INTERFACE ITF_CyclicUpdate

// Uses HRESULT outputs for management of different scenarios, such as errors and non-completes

//    0 - No Output / Execute In Progress
//    1 - Execute Complete
//    2 - Execute Failed, No Program Error, Object's Internal Timer Exceeded Limit.
//   -1 - Execute Failed, Program Error

METHOD CyclicUpdate : HRESULT

// Uses HRESULT outputs for management of different scenarios, such as errors and non-completes

//    0 - No Output / Execute In Progress
//    1 - Execute Complete
//    2 - Execute Failed, No Program Error, Object's Internal Timer Exceeded Limit.
//   -1 - Execute Failed, Program Error
END_METHOD

END_INTERFACE

(* stored: Version 1.1.0.1, ProductVersion 3.1.4024.12
   Itf ITF_CyclicUpdate: Id {90bd103a-7016-4ff7-8d58-86cc61bdd8ac}
   Method CyclicUpdate: Id {30e66b99-5a80-463a-bcbf-e44a06ca53a7} *)
